KUKA KRL data list: SetCamada.dat

&ACCESS RVO
&REL 3
&PARAM EDITMASK = *
DEFDAT  SetCamada

ENDDAT
